DATA_BLOCK "ST10_Flow15_FRobot_3_iDB"
{ S7_Optimized_Access := 'TRUE' }
VERSION : 0.1
NON_RETAIN
// ATTRIBUTES
// AUTO_NUMBER = False
// BLOCK_NUMBER = 1085
// END_ATTRIBUTES
"ST10_Flow15_FRobot_3"

BEGIN

END_DATA_BLOCK

